TYPE ST_StationData :
STRUCT
	Status		: INT;
	VisuPosX 	: INT;
	VisuPosY 	: INT;
//	ProcessTimeAve	: TIME :=T#1S;		// average station process time
//	ProcessTimeAct	: TIME;				// actual (randomized) process time
	
END_STRUCT
END_TYPE

(* stored: Version 1.1.0.1, ProductVersion 3.1.4024.12
   DUT ST_StationData: Id {073477ec-8f7d-4a9c-8ada-62ba498f2634} *)
